ABB RAPID module: mSettings_Spindle.sys

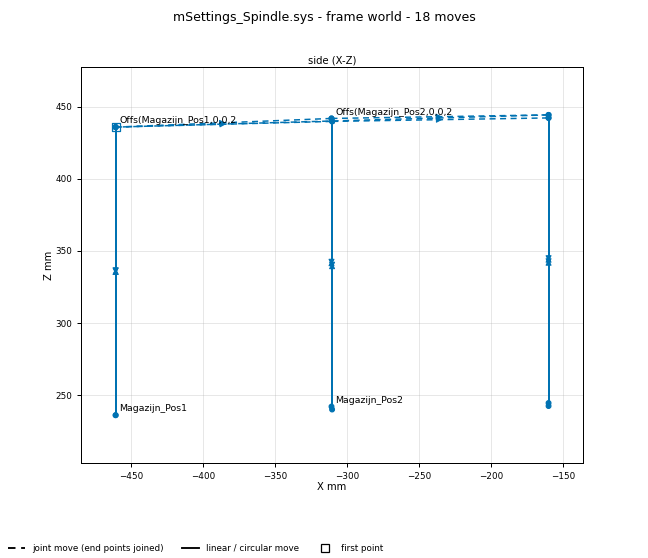
[picture p0: tool path of mSettings_Spindle.sys in frame world, 18 of 35 moves have a stored position in this frame; points joined in program order, loops and branches not executed]
MODULE mSettings_Spindle(SYSMODULE)
    !toolmagazijn
    CONST num EmptySpindel :=0;
    CONST num Boor_11m := 1;
    CONST num Frees := 2;
    CONST num Frees_13 := 3;
    CONST num empty4 := 4;
    CONST num empty5 := 5;
    CONST num empty6 := 6;
    local PERS bool  bActiveTool{6} := [FALSE,TRUE,FALSE,FALSE,FALSE,FALSE];
    !joint targets
    CONST jointtarget pHomeJoint_spindel:=[[-114.954,-13.8901,3.19333,84.0191,-65.7533,-33.8858],[500.019,9E+09,9E+09,9E+09,9E+09,9E+09]];
    !Robtargets
    local CONST robtarget Magazijn_Pos1:=[[-460.63,-1000.68,236],[0.00362869,-0.999994,0.000227334,-0.00060485],[-2,0,-1,0],[500.003,9E+09,9E+09,9E+09,9E+09,9E+09]];
    local CONST robtarget Magazijn_Pos2:=[[-310.78,-1003.15,242],[0.00365054,-0.999993,0.000240162,-0.000632287],[-2,0,-1,0],[500.006,9E+09,9E+09,9E+09,9E+09,9E+09]];
    local CONST robtarget Magazijn_Pos3:=[[-160.10,-1003.44,244.47],[0.00364503,-0.999993,0.000235225,-0.000610413],[-2,0,-1,0],[500.002,9E+09,9E+09,9E+09,9E+09,9E+09]];
    local CONST robtarget Magazijn_Pos4:=[[-460.63,-1000.68,235.99],[0.00362869,-0.999994,0.000227334,-0.00060485],[-2,0,-1,0],[500.003,9E+09,9E+09,9E+09,9E+09,9E+09]];
    local CONST robtarget Magazijn_Pos5:=[[-310.37,-1002.67,239.95],[0.00363142,-0.999993,0.00022822,-0.000658208],[-2,0,-1,0],[500.001,9E+09,9E+09,9E+09,9E+09,9E+09]];
    local CONST robtarget Magazijn_Pos6:=[[-160.10,-1003.45,242.36],[0.00363494,-0.999994,0.000227547,-0.000607041],[-2,0,-1,0],[500.003,9E+09,9E+09,9E+09,9E+09,9E+09]];
    !Wobjdata
    TASK PERS wobjdata wobj_Magazijn:=[FALSE,TRUE,"",[[0,0,0],[1,0,0,0]],[[0,0,0],[1,0,0,0]]];
    !Tooldata
    TASK PERS tooldata tSpindle:=[TRUE,[[314,-0.75,111],[0.707107,0,0.707107,0]],[25.8,[102.9,49.8,-410.4],[1,0,0,0],0,0,0]];
    TASK PERS tooldata tSpindleSensor:=[TRUE,[[437.094,57.5763,-0.711741],[0.707107,0,0.707107,0]],[25.8,[102.9,49.8,-410.4],[1,0,0,0],0,0,0]];
    TASK PERS tooldata boor_11mm_L190:=[TRUE,[[502,-0.75,111],[0.707107,0,0.707107,0]],[25.8,[102.9,49.8,-410.4],[1,0,0,0],0,0,0]];
    TASK PERS tooldata tFrees_10:=[TRUE,[[505,-0.75,111],[0.707107,0,0.707107,0]],[25.8,[102.9,49.8,-410.4],[1,0,0,0],0,0,0]];
    TASK PERS tooldata tFrees_13:=[TRUE,[[515,-0.75,111],[0.707107,0,0.707107,0]],[25.8,[102.9,49.8,-410.4],[1,0,0,0],0,0,0]];

    !Speedata
    PERS speeddata vBoren_11_190:=[4,500,5000,1000];
    PERS speeddata vBoren_aanzet:=[10,500,5000,1000];

    PERS speeddata vFrezen:=[15,500,5000,1000];
    PERS speeddata vBorenMetFrees:=[4,500,5000,1000];
    PERS speeddata vFrees_aanzet:=[80,500,5000,1000];

    !counter to keep trqck of oil pusle,
    PERS num nOilPulses := 1;

    LOCAL PROC rInitSpindelData()
        !voorlopig gefoefel
        TEST fGet_activeTool()
          CASE 1:
             vBoren_11_190 := Spindeltool{1}.VoedingBoren;
             vBoren_aanzet := Spindeltool{1}.VoedingAanzetBoren;
          CASE 2:
             vBoren_11_190 := Spindeltool{2}.VoedingBoren;
             vBoren_aanzet := Spindeltool{2}.VoedingAanzetBoren;
             vFrezen := Spindeltool{2}.VoedingFrezen;
             vBorenMetFrees := Spindeltool{2}.VoedingBoren;
             vFrees_aanzet := Spindeltool{2}.VoedingAanzetFrezen;
          CASE 3:
             vBoren_11_190 := Spindeltool{3}.VoedingBoren;
             vBoren_aanzet := Spindeltool{3}.VoedingAanzetBoren;
             vFrezen := Spindeltool{3}.VoedingFrezen;
             vBorenMetFrees := Spindeltool{3}.VoedingBoren;
             vFrees_aanzet := Spindeltool{3}.VoedingAanzetFrezen;
         DEFAULT:
           !do nothing
        ENDTEST
    ENDPROC

    LOCAL PROC rteach_mag_Pos()
    !***************************************
    ! Proc: rteach_mag_Pos
    ! Description: om posities in magazijn te teachen
    !***************************************
        Stop;
        MoveJ Offs(Magazijn_Pos1,0,0,200),v200,fine,tSpindle\WObj:=wobj_Magazijn;
        MoveL Magazijn_Pos1,v10,fine,tSpindle\WObj:=wobj_Magazijn;
        MoveL Offs(Magazijn_Pos1,0,0,200),v200,fine,tSpindle\WObj:=wobj_Magazijn;
        Stop;
        MoveJ Offs(Magazijn_Pos2,0,0,200),v200,fine,tSpindle\WObj:=wobj_Magazijn;
        MoveL Magazijn_Pos2,v10,fine,tSpindle\WObj:=wobj_Magazijn;
        MoveL Offs(Magazijn_Pos2,0,0,200),v200,fine,tSpindle\WObj:=wobj_Magazijn;
        Stop;
        MoveJ Offs(Magazijn_Pos3,0,0,200),v200,fine,tSpindle\WObj:=wobj_Magazijn;
        MoveL Magazijn_Pos3,v10,fine,tSpindle\WObj:=wobj_Magazijn;
        MoveL Offs(Magazijn_Pos3,0,0,200),v200,fine,tSpindle\WObj:=wobj_Magazijn;
        Stop;
        MoveJ Offs(Magazijn_Pos4,0,0,200),v200,fine,tSpindle\WObj:=wobj_Magazijn;
        MoveL Magazijn_Pos4,v10,fine,tSpindle\WObj:=wobj_Magazijn;
        MoveL Offs(Magazijn_Pos4,0,0,200),v200,fine,tSpindle\WObj:=wobj_Magazijn;
        Stop;
        MoveJ Offs(Magazijn_Pos5,0,0,200),v200,fine,tSpindle\WObj:=wobj_Magazijn;
        MoveL Magazijn_Pos5,v10,fine,tSpindle\WObj:=wobj_Magazijn;
        MoveL Offs(Magazijn_Pos5,0,0,200),v200,fine,tSpindle\WObj:=wobj_Magazijn;
        Stop;
        MoveJ Offs(Magazijn_Pos6,0,0,200),v200,fine,tSpindle\WObj:=wobj_Magazijn;
        MoveL Magazijn_Pos6,v10,fine,tSpindle\WObj:=wobj_Magazijn;
        MoveL Offs(Magazijn_Pos6,0,0,200),v200,fine,tSpindle\WObj:=wobj_Magazijn;
        Stop;
        !
    ENDPROC

    PROC Set_Tool_Manual()
    !***************************************
    ! Proc: Set_Tool_Manual
    ! Description: manueel tool actief zetten
    !***************************************
        var num selectedTool;
        selectedTool := fSelect_tool();
        ! set selected tool active
        FOR i FROM 1 TO 6 STEP 1 DO
           IF i = selectedTool THEN
             bActiveTool{i} := TRUE;
           ELSE
             bActiveTool{i} := FALSE;
           ENDIF
        ENDFOR
    ENDPROC

    LOCAL FUNC num fSelect_tool()
    !***************************************
    ! Func: fSelect_tool
    ! Description: manueel tool selecteren
    !***************************************
        VAR btnres nAnswer;
        lbl_1:
            nAnswer:=UIMessageBox(\Header:="Welke spindel tool?",\BtnArray:=[Spindeltool{1}.toolnaam,Spindeltool{2}.toolnaam,Spindeltool{3}.toolnaam,"","MEER"]);
            IF nAnswer > 3 THEN
              nAnswer:=UIMessageBox(\Header:="Welke spindel tool?",\BtnArray:=[Spindeltool{4}.toolnaam,Spindeltool{5}.toolnaam,Spindeltool{6}.toolnaam,"GeenTool","MEER"]);
              IF nAnswer = 5 THEN
                GOTO lbl_1;
              ELSEIF nAnswer = 4 THEN
                 !no tool
                 nAnswer := 0;
              ELSE
                 nAnswer := nAnswer + 3;
              ENDIF
            ENDIF
            TPWrite("User selected:"+ NumToStr(nAnswer,0) + " Active:" + NumToStr(fGet_activeTool(),0));
            RETURN nAnswer;
    ENDFUNC

    PROC Get_tool_Manual()
    !***************************************
    ! Proc: Get_tool_Manual
    ! Description: manueel tool wisselen
    !***************************************
     Set_Tool(fSelect_tool());
     !
    ENDPROC

    PROC Check_Tool(num nTool)
    !***************************************
    ! Proc: Check_Tool
    ! Description: check if tool is active
    !***************************************
        VAR btnres nAnswer;
        VAR num nActieve_Tool;
        nActieve_Tool := fGet_activeTool();
        IF NOT nTool = nActieve_Tool THEN
         WHILE TRUE DO
          nAnswer := UIMessageBox(\Header:="Magazijn fout"\MsgArray:=["fout tool actief !","ga manueel om tool"],\BtnArray:=["","","","","OK"]);
         ENDWHILE
        ENDIF
    !
    ENDPROC

    PROC Set_Tool(num nTool)
    !***************************************
    ! Proc: Set_Tool
    ! Description: get selected spindel tool
    !***************************************
        VAR num nActieve_Tool;
        nActieve_Tool := fGet_activeTool();
        PDispOff;
        EOffsOff;
        !put gripper away take dummy
        Set_Gripper(DummyTool);
        !
        IF NOT nActieve_Tool = nTool THEN
          MoveAbsJ fArm_only(pHomeJoint_spindel)\NoEOffs, v4000, z50, tSpindle;
          MoveAbsJ pHomeJoint_spindel\NoEOffs, v4000, z50, tSpindle;
          IF NOT nActieve_Tool = 0 THEN
            rStop_Spindle;
            rDetach_tool nActieve_Tool;
          ENDIF
          IF NOT nTool = 0 THEN
           rAttach__tool nTool;
          ENDIF
          MoveAbsJ pHomeJoint_spindel\NoEOffs, v4000, z50, tSpindle;
        ENDIF
        !
    ENDPROC

    LOCAL FUNC num fGet_activeTool()
    !***************************************
    ! Func: fGet_activeTool
    ! Description: checks if tested tool is active
    !***************************************
    VAR num nActiveTool := 0;
    VAR bool bFoundActivetool := false;
    VAR btnres nAnswer;

    FOR i FROM 1 TO 6 STEP 1 DO
      IF bActiveTool{i} THEN
         nActiveTool := i;
         IF NOT bFoundActivetool THEN
          bFoundActivetool := TRUE;
         ELSE
            nAnswer := UIMessageBox(\Header:="Magazijn fout"\MsgArray:=["meer dan 1 tool actief !","bevestig manueel de active tool"],\BtnArray:=["","","","","Selecteer"]);
            Set_Tool_Manual;
         ENDIF
      ENDIF
    ENDFOR

    RETURN nActiveTool;
    ENDFUNC

    LOCAL FUNC robtarget fToolMagpos(num nTool)
    !***************************************
    ! FUNC: fToolMagpos
    ! Description: gets tool mag pos by idx
    !***************************************
      TEST nTool
        CASE 1:
           RETURN Magazijn_Pos1;
        CASE 2:
           RETURN Magazijn_Pos2;
        CASE 3:
           RETURN Magazijn_Pos3;
        CASE 4:
           RETURN Magazijn_Pos4;
        CASE 5:
           RETURN Magazijn_Pos5;
        CASE 6:
           RETURN Magazijn_Pos6;
        DEFAULT:
            EXIT;
        ENDTEST
    ENDFUNC

   LOCAL PROC rDetach_tool(num Toolnum)
    !***************************************
    ! Proc: rDetach_tool
    ! Description: drop tool in mag pos
    !***************************************
        VAR robtarget Magpos;
        Magpos := fToolMagpos(Toolnum);
        !
            Movej Offs(Magpos,0,0,200),v7000,fine,tSpindleSensor\WObj:=wobj_Magazijn;
            !check no tool present (deep check)
            MoveL Offs(Magpos,0,0,40),v500,fine,tSpindleSensor\WObj:=wobj_Magazijn;
            WaitTime \InPos, 2;
            CheckInput di_SpindelSensor,0, \CheckTimeOut:=3,"Tool magazijn niet leeg! ";
            Movel Offs(Magpos,0,0,200),v1000,fine,tSpindle\WObj:=wobj_Magazijn;
            MoveL Offs(Magpos,0,0,20),v500,z0,tSpindle\WObj:=wobj_Magazijn;
            MoveL Offs(Magpos,0,0,2),v50,fine,tSpindle\WObj:=wobj_Magazijn;
            rSpindle_Unlock;
            bActiveTool{Toolnum} :=FALSE;
            MoveL Offs(Magpos,0,0,200),v200,fine,tSpindle\WObj:=wobj_Magazijn;
            Reset doSpindle_Air_On;
            !check tool detached
            MoveL Offs(Magpos,-5,0,68),v500,fine,tSpindleSensor\WObj:=wobj_Magazijn;
            CheckInput di_SpindelSensor,1, \CheckTimeOut:=3,"Tool hangt nog aan robot! ";
            MoveL Offs(Magpos,0,0,200),v1000,fine,tSpindle\WObj:=wobj_Magazijn;
        !
    ENDPROC

   LOCAL PROC rAttach__tool( num Toolnum)
    !***************************************
    ! Proc: rAttach__tool
    ! Description: get tool in mag pos
    !***************************************
        VAR robtarget Magpos;
        Magpos := fToolMagpos(Toolnum);
        !
            Movej Offs(Magpos,0,0,200),v500,fine,tSpindleSensor\WObj:=wobj_Magazijn;
            !check  tool present
            MoveL Offs(Magpos,-5,0,68),v500,fine,tSpindleSensor\WObj:=wobj_Magazijn;
            CheckInput di_SpindelSensor,1, \CheckTimeOut:=3,"Tool niet aanwezig in magazijn! ";
            rSpindle_Unlock;
            MoveL Offs(Magpos,0,0,100),v500,z0,tSpindle\WObj:=wobj_Magazijn;
            MoveL Magpos,v50,fine,tSpindle\WObj:=wobj_Magazijn;
            rSpindle_Lock;
            bActiveTool{Toolnum} :=TRUE;
            MoveL Offs(Magpos,0,0,100),v200,fine,tSpindle\WObj:=wobj_Magazijn;
            MoveL Offs(Magpos,0,0,200),v1000,fine,tSpindle\WObj:=wobj_Magazijn;
        !
    ENDPROC


    LOCAL PROC rSpindle_Unlock()
    !***************************************
    ! Proc: rSpindle_Unlock
    ! Description: unlock spindel
    !***************************************
        SetDO doSpindle_Air_On,0;
        SetDO doSpindle_Release,1;
        CheckInput diSpindle_S2,1, \CheckTimeOut:=3,"Sinpdel sensor fout diSpindle_S2 0 ";
        CheckInput diSpindle_S3,0, \CheckTimeOut:=3,"Sinpdel sensor fout diSpindle_S3 1 ";
        CheckInput diSpindle_S4,0, \CheckTimeOut:=3,"Sinpdel sensor fout diSpindle_S4 1 ";
        !
    ENDPROC

    LOCAL PROC rSpindle_Lock()
    !***************************************
    ! Proc: rSpindle_Lock
    ! Description: lock spindel
    !***************************************
        SetDO doSpindle_Air_On,1;
        SetDO doSpindle_Release,0;
        CheckInput diSpindle_S2,0,  \CheckTimeOut:=3,"Sinpdel sensor fout diSpindle_S2 1 ";
        CheckInput diSpindle_S3,1, \CheckTimeOut:=3,"Sinpdel sensor fout diSpindle_S3 2 ";
        CheckInput diSpindle_S4,1, \CheckTimeOut:=5,"Sinpdel sensor fout diSpindle_S4 0 ";
        !
    ENDPROC

    PROC rStart_Spindle(\num nSpeed)
    !***************************************
    ! Proc: rStart_Spindle
    ! Description: start spindel
    ! nSpeed wil override default toolspeed
    !***************************************
       VAR bool bAlreadyOn;
       IF DOutput(so_Boren_aan) = 1 THEN
           bAlreadyOn := true;
        ENDIF

        rInitSpindelData;
        Set doSpindle_Air_On; !moet anders draait hij stroef !
        Set so_Boren_aan;
        IF Present(nSpeed) THEN
         SetAO aoPLC_Spindle_Speed,nSpeed;
        ELSE
         SetAO aoPLC_Spindle_Speed,Spindeltool{fGet_activeTool()}.Toerental;
        ENDIF
        IF (bAlreadyOn = FALSE) THEN
         rCheckSpindelRunning \nPulses:=3;
        ENDIF
        rSpindelSprVsn TRUE \init ;
        !
    ENDPROC

   PROC rOilPulse(\num nPulseTime, \switch keepON )
    !***************************************
    ! Proc: rOil
    ! Description: control oil mister
    !***************************************
    SetDO doSpindle_CoolingAir_On, 1;
    SetDO so_Olie_aan, 0;

   IF Present(nPulseTime) THEN
    PulseDO \PLength:= nPulseTime, doSpindle_CoolingAir_On;
    PulseDO \High \PLength:= nPulseTime, so_Olie_aan;
   ELSE
       IF Present(keepOn) THEN
         SetDO doSpindle_CoolingAir_On, 0;
         SetDO so_Olie_aan, 1;
       else
        PulseDO \PLength:= 2, doSpindle_CoolingAir_On;
        PulseDO \High \PLength:= 2, so_Olie_aan;
       ENDIF
   ENDIF


   ENDPROC

   PROC roilOFF()
    !***************************************
    ! Proc: roilOFF
    ! Description: interupt oil mister
    !***************************************
      SetDO so_Olie_aan, 0;
      SetDO doSpindle_CoolingAir_On, 1;
   ENDPROC

    PROC roiliNIT()
    !***************************************
    ! Proc: roilOFF
    ! Description: interupt oil mister
    !***************************************
     nOilPulses := 10000;
   ENDPROC

  PROC rAutoOilPulse(\num nPulseTime, \switch keepON, \num nPulseinterval)
    !***************************************
    ! Proc: rOilnPulseinterval
    ! Description: control oil mister witch counter
    !***************************************
VAR num lPulsinterval;
   IF NOT Present(nPulseinterval) THEN
    lPulsinterval := 5;
   ELSE
    lPulsinterval := nPulseinterval;
   ENDIF
   IF nOilPulses >= lPulsinterval THEN
     rOilPulse \nPulseTime?nPulseTime, \keepON?keepON;
     nOilPulses := 0;
   ELSE
    Incr nOilPulses;
    roilOFF;
   ENDIF
 ENDPROC

    PROC rStop_Spindle()
    !***************************************
    ! Proc: rStop_Spindle
    ! Description: stop spindel
    !***************************************
        rSpindelSprVsn FALSE;
        SetAO aoPLC_Spindle_Speed,0;
        Reset so_Boren_aan;
        Reset doSpindle_Air_On;
        Reset so_Olie_aan;
        !
    ENDPROC

    PROC rWait_Spindel()
    !***************************************
    ! Proc: rWait_Spindel
    ! Description: wait for spindle to get rpm
    ! Connected in eventroutine and trap
    !***************************************
       IF  DOutput(so_Boren_aan) = 1 THEN
           rCheckSpindelRunning \nPulses:=3;
       ENDIF
    ENDPROC

    local PROC rSpindelSprVsn(bool bEnable \switch init)
    !***************************************
    ! Trap: tSpindelSprVsn
    ! Description: supervision for spindle
    ! check if spindel is not stopped
    !***************************************
     IF Present(init) THEN
      IDelete Int1SprvSpindel;
      CONNECT Int1SprvSpindel WITH tSpindelSprVsn;
      ISignalDI di_SpindleDriveOK,0,Int1SprvSpindel;
      ISleep Int1SprvSpindel;
     ENDIF

     IF bEnable THEN
      IWatch Int1SprvSpindel;
     ELSE
      !ISleep Int1SprvSpindel;
     ENDIF
    ENDPROC

  TRAP tSpindelSprVsn
    !***************************************
    ! Trap: tSpindelSprVsn
    ! Description: Supervision trap that
    ! stops robot with alarm message
    ! Connected in rSpindelSprVsn
    !***************************************
   VAR btnres nAnswer;
   ISleep Int1SprvSpindel;
   StopMove;
   StorePath;
   nAnswer := UIMessageBox(\Header:="Spindelfout"\MsgArray:=["Spindel onverwachts gestopt","controleer dat de spindle vrij kan draaien","controleer of de spindle drive oke is"],\BtnArray:=["","","","","Reset"]);
   RestoPath;
   IWatch Int1SprvSpindel;
   StartMove;
   rWait_Spindel;
  ENDTRAP


  PROC rCheckSpindelRunning(\Num nPulses)
    !***************************************
    ! Trap: rCheckSpindelRunning
    ! Description: kijk of spindel draait aan de hand van pulsen
    !***************************************
   VAR btnres nAnswer;
   VAR num nPulscount;
   VAR bool bTimeout;
   VAR dionum nFlipstate;
   lblreset:
       nFlipstate := DInput(diSpindle_No_Rotation);
       IF NOT Present(nPulses) THEN
           nPulses := 3;
       ENDIF
       FOR i FROM 1 TO nPulses DO
           IF DOutput(so_Boren_aan) = 1 then
               WaitDI diSpindle_No_Rotation, nFlipstate \MaxTime:=3000 \Timeflag := bTimeout;
               IF bTimeout THEN
                 Stop;
                 nAnswer := UIMessageBox(\Header:="Spindelfout"\MsgArray:=["Spindel onverwachts gestopt","controleer dat de spindle vrij kan draaien"],\BtnArray:=["","","","","Reset"]);
                 GOTO lblreset;
               ENDIF
               !
               IF nFlipstate = 1 THEN
                  nFlipstate:= 0;
               ELSE
                  nFlipstate :=1;
               ENDIF
           ENDIF
       ENDFOR
  ENDPROC
ENDMODULE
